FUNCTION_BLOCK TN_INPUT_EDIT_LINE
VAR
	in_count : INT;
	in_Count_End : INT;
	in_CursorOffset : INT;
	by_Attr : BYTE;
	st_String : STRING;
	bo_Pos_Found : BOOL;
	st_CHAR : STRING(1);
	in_old_charpos : INT;
END_VAR
VAR
	FB_TN_SC_WRITE : TN_SC_WRITE;
END_VAR
VAR_IN_OUT
	Xus_TN_SCREEN : us_TN_SCREEN;
	Xus_TN_INPUT_CONTROL_DATA : us_TN_INPUT_CONTROL_DATA;
END_VAR

(*
version 1.0		10. mai 2010
programmer		ks
tested by		ks

TN_INPUT_EDIT_LINE ermöglicht die Eingabe von Texten durch eine Editierbare Eingabezeile
*)

(* Cursorsteuerung rücksetzen *)
in_CursorOffset := INT#0;

IF Xus_TN_INPUT_CONTROL_DATA.bo_Focus = TRUE THEN

	(* Texteingabe erkannt ? *)
	IF Xus_TN_INPUT_CONTROL_DATA.by_Input_ASCII_Code > BYTE#0 THEN

		IF (Xus_TN_INPUT_CONTROL_DATA.bo_Input_Only_Num = TRUE AND Xus_TN_INPUT_CONTROL_DATA.bo_Input_ASCII_IsNum = TRUE)
			OR (Xus_TN_INPUT_CONTROL_DATA.bo_Input_Only_Num = FALSE) THEN

			(* ASCII Wert in einen String wandeln *)
			st_CHAR := CHR_TO_STRING(C:=Xus_TN_INPUT_CONTROL_DATA.by_Input_ASCII_Code);

			(* Eingabe übernehmen *)
			Xus_TN_INPUT_CONTROL_DATA.st_Input_Data := REPLACE(Xus_TN_INPUT_CONTROL_DATA.st_Input_Data,
			st_CHAR,INT#1,Xus_TN_INPUT_CONTROL_DATA.in_Cursor_Pos);

			in_CursorOffset := INT#1;
			Xus_TN_INPUT_CONTROL_DATA.bo_Update_Input := TRUE;
		END_IF;
	END_IF;

	CASE BYTE_TO_INT(Xus_TN_INPUT_CONTROL_DATA.by_Input_Exten_Code) OF

	67: (* Cursor rechts gedrückt *)
		in_CursorOffset := INT#1;

	68: (* Cursor links gedrückt *)
		in_CursorOffset := -1;

	08: (* Backspace gedrückt *)
		Xus_TN_INPUT_CONTROL_DATA.st_Input_Data := REPLACE(Xus_TN_INPUT_CONTROL_DATA.st_Input_Data, ' ', 1,Xus_TN_INPUT_CONTROL_DATA.in_Cursor_Pos);
		Xus_TN_INPUT_CONTROL_DATA.bo_Update_Input := TRUE;
		in_CursorOffset := -1;

	13: (* Enter-Taste gedrückt *)
		IF LEN(Xus_TN_INPUT_CONTROL_DATA.st_Input_Mask) > INT#00 THEN
			(* Eingabestring übernehmen *)
			Xus_TN_INPUT_CONTROL_DATA.st_Input_String := Xus_TN_INPUT_CONTROL_DATA.st_Input_Data;

			(* Eingabestring -> links und rechts Leerzeichen entfernen *)
			Xus_TN_INPUT_CONTROL_DATA.st_Input_String := TRIME(str:=Xus_TN_INPUT_CONTROL_DATA.st_Input_String);
			Xus_TN_INPUT_CONTROL_DATA.bo_Input_Entered := TRUE;

			(* neue Eingabe vorbereiten *)
			Xus_TN_INPUT_CONTROL_DATA.st_Input_Data := Xus_TN_INPUT_CONTROL_DATA.st_Input_Mask;

			Xus_TN_INPUT_CONTROL_DATA.in_Cursor_Pos := INT#1;
			Xus_TN_INPUT_CONTROL_DATA.bo_Update_Input := TRUE;

			(* suche erstes Position in Eingabemaske *)
			st_CHAR := MID(Xus_TN_INPUT_CONTROL_DATA.st_Input_Mask,1,Xus_TN_INPUT_CONTROL_DATA.in_Cursor_Pos);
			IF st_CHAR <> ' ' THEN
				(* nächsten Eingabeposition suchen *)
				in_CursorOffset := INT#1;
			END_IF;
		END_IF;
	END_CASE;
END_IF;

(* Cursor richtung rechts bewegen                                   *)
IF (in_CursorOffset > INT#0) OR (Xus_TN_INPUT_CONTROL_DATA.in_Cursor_Pos = INT#0) THEN
	bo_Pos_Found := FALSE;

	in_Count := Xus_TN_INPUT_CONTROL_DATA.in_Cursor_Pos + INT#1;
	in_Count_End := LEN(Xus_TN_INPUT_CONTROL_DATA.st_Input_Mask);

	WHILE (in_count <= in_Count_End) AND (bo_Pos_Found = FALSE) DO

		st_CHAR := MID(Xus_TN_INPUT_CONTROL_DATA.st_Input_Mask,1,in_count);
		IF st_CHAR = ' ' THEN
			Xus_TN_INPUT_CONTROL_DATA.in_Cursor_Pos := in_count;
			Xus_TN_INPUT_CONTROL_DATA.bo_Update_Input := TRUE;
			bo_Pos_Found := TRUE;
		END_IF;

		in_count := in_count + INT#1;

	END_WHILE;
END_IF;

(* Cursor richtung links bewegen *)
IF in_CursorOffset < INT#0 THEN
	bo_Pos_Found := FALSE;

	in_Count     := Xus_TN_INPUT_CONTROL_DATA.in_Cursor_Pos - INT#01;
	in_Count_End := INT#1;

	WHILE (in_count >= in_Count_End) AND (bo_Pos_Found = FALSE) DO

		st_CHAR := MID(Xus_TN_INPUT_CONTROL_DATA.st_Input_Mask,1,in_count);
		IF st_CHAR = ' ' THEN
			Xus_TN_INPUT_CONTROL_DATA.in_Cursor_Pos := in_count;
			Xus_TN_INPUT_CONTROL_DATA.bo_Update_Input := TRUE;
			bo_Pos_Found := TRUE;
		END_IF;

		in_count := in_count - INT#1;
	END_WHILE;
END_IF;

(* maximale Cursorposition ? *)
IF Xus_TN_INPUT_CONTROL_DATA.in_Cursor_Pos > LEN(Xus_TN_INPUT_CONTROL_DATA.st_Input_Data) THEN
	Xus_TN_INPUT_CONTROL_DATA.in_Cursor_Pos := LEN(Xus_TN_INPUT_CONTROL_DATA.st_Input_Data);
	Xus_TN_INPUT_CONTROL_DATA.bo_Update_Input := TRUE;
END_IF;

(* minimale Cursorposition ? *)
IF Xus_TN_INPUT_CONTROL_DATA.in_Cursor_Pos < INT#1 THEN
	Xus_TN_INPUT_CONTROL_DATA.in_Cursor_Pos := INT#1;
	Xus_TN_INPUT_CONTROL_DATA.bo_Update_Input := TRUE;
END_IF;

(* Aktualisierung der Anzeige *)
IF (Xus_TN_INPUT_CONTROL_DATA.bo_Update_Input = TRUE) OR (Xus_TN_INPUT_CONTROL_DATA.bo_Update_All = TRUE) THEN

	(* Title-Text ausgeben *)
	IF (Xus_TN_INPUT_CONTROL_DATA.bo_Update_All = TRUE) THEN

		IF (Xus_TN_INPUT_CONTROL_DATA.in_Title_X_Offset = INT#00) AND (Xus_TN_INPUT_CONTROL_DATA.in_Title_Y_Offset = INT#00) THEN
			(* wenn Offset X,Y =0 dann Titlestring links vom Element positionieren *)
			FB_TN_SC_WRITE.Iin_Y := Xus_TN_INPUT_CONTROL_DATA.in_Y;
			FB_TN_SC_WRITE.Iin_X := Xus_TN_INPUT_CONTROL_DATA.in_X - LEN(Xus_TN_INPUT_CONTROL_DATA.st_Title_String);
		ELSE
			(* Title-Text durch Row, Color-Offset ausgeben *)
			FB_TN_SC_WRITE.Iin_Y := Xus_TN_INPUT_CONTROL_DATA.in_Y + Xus_TN_INPUT_CONTROL_DATA.in_Title_Y_Offset;
			FB_TN_SC_WRITE.Iin_X := Xus_TN_INPUT_CONTROL_DATA.in_X + Xus_TN_INPUT_CONTROL_DATA.in_Title_X_Offset;
		END_IF;

		(* Title-Text durch Row, Color-Offset ausgeben *)
		FB_TN_SC_WRITE(	Iby_ATTR := Xus_TN_INPUT_CONTROL_DATA.by_Title_Attr,
						Ist_STRING := Xus_TN_INPUT_CONTROL_DATA.st_Title_String,
						Xus_TN_SCREEN := Xus_TN_SCREEN);
	END_IF;

	(* Eingabetext ausgeben *)
	IF (Xus_TN_INPUT_CONTROL_DATA.bo_Input_Hidden = TRUE) THEN

		st_String := '';

		IF LEN(Xus_TN_INPUT_CONTROL_DATA.st_Input_Data) = LEN(Xus_TN_INPUT_CONTROL_DATA.st_Input_Mask) THEN
			(* Eingabemodus: HIDDEN *)
			FOR in_count := 1 TO LEN(Xus_TN_INPUT_CONTROL_DATA.st_Input_Data) DO

				(* Zeichen aus Eingabemaske lesen *)
				st_CHAR := MID(Xus_TN_INPUT_CONTROL_DATA.st_Input_Mask,1,in_count);

				(* Eingabe oder Maskenzeichen ausgeben *)
				IF st_CHAR = ' ' THEN

					(* Zeichen aus Eingabedata lesen *)
					st_CHAR := MID(Xus_TN_INPUT_CONTROL_DATA.st_Input_Data,1,in_count);

					IF st_CHAR = ' ' THEN
						(* Leerzeichen ausgeben *)
						st_String := CONCAT(st_String, ' ');

					ELSE
						(* verdecktes Zeichen ausgeben *)
						st_String := CONCAT(st_String, '*');

					END_IF;

				ELSE
					(* Zeichen aus Eingabemaske übernehmen *)
					st_CHAR := MID(Xus_TN_INPUT_CONTROL_DATA.st_Input_Data,1,in_count);
					st_String := CONCAT(st_String,st_CHAR);

				END_IF;
			END_FOR;
		END_IF;
	ELSE

		(* Eingabemodus: NORMAL *)
		st_String := Xus_TN_INPUT_CONTROL_DATA.st_Input_Data;

	END_IF;

	(* String ausgeben *)

	IF Xus_TN_INPUT_CONTROL_DATA.bo_Focus = TRUE THEN
		by_Attr := Xus_TN_INPUT_CONTROL_DATA.by_Attr_mF;
	ELSE
		by_Attr := Xus_TN_INPUT_CONTROL_DATA.by_Attr_oF;
	END_IF;

	FB_TN_SC_WRITE(	Iin_Y := Xus_TN_INPUT_CONTROL_DATA.in_Y,
					Iin_X := Xus_TN_INPUT_CONTROL_DATA.in_X,
					Iby_ATTR := by_Attr,
					Ist_STRING := st_String,
					Xus_TN_SCREEN := Xus_TN_SCREEN);

	(* Cursor auf aktuelle Position setzen *)
	Xus_TN_INPUT_CONTROL_DATA.in_Cursor_Y := Xus_TN_INPUT_CONTROL_DATA.in_Y;
	Xus_TN_INPUT_CONTROL_DATA.in_Cursor_X := Xus_TN_INPUT_CONTROL_DATA.in_X + Xus_TN_INPUT_CONTROL_DATA.in_Cursor_Pos - INT#1;

	in_old_charpos := INT#0;

	(* Update-Flag's rücksetzen *)
	Xus_TN_INPUT_CONTROL_DATA.bo_Update_All := FALSE;
	Xus_TN_INPUT_CONTROL_DATA.bo_Update_Input := FALSE;
END_IF;

(* revision history
ks	10. mai. 2010	rev 1.0
	original version
*)

END_FUNCTION_BLOCK

(* stored: Version 1.1.0.1, ProductVersion 3.1.4022.7
   POU TN_INPUT_EDIT_LINE: Id {dc319b35-a3c3-4a76-957b-d022e76301a4}, SpecialFunc None *)
